(* PLC project Generated.project, CODESYS CODESYS V3.5 SP19 Patch 1 *)
(* stored: creationDateTime 2026-09-06T13:00:42.484991, modificationDateTime 2026-09-06T13:00:42.484991 *)

TYPE ST_Chain_Winch_Safety : STRUCT
  Idx301_EmergencyChainClosed : BOOL;  (* 1 = Boucle Urgence OK (Armé) | 0 = Arrêt d'Urgence Appuyé *)
  Idx302_SafeStopActive : BOOL;  (* 0 = Sain (Autorisé) | 1 = Arrêt Rapide Métier Actif *)
  Idx303_PowerCutOffActive : BOOL;  (* 0 = Puissance OK | 1 = Coupure Puissance Sécurité *)
  Idx304_TopSensorPhysical_DI : BOOL;  (* 1 = Capteur Haut Libre (Sain) | 0 = Butée Haute Atteinte *)
  Idx305_TopSensorBypassActive : BOOL;  (* 0 = Capteur Actif | 1 = Capteur Haut Shunté IHM ⚠️ *)
  Idx306_AscentPermitEffective : BOOL;  (* 1 = Ascending Autorisée | 0 = ASCENDING BLOQUÉE *)
  Idx307_SlackCablePhysical_DI : BOOL;  (* 1 = Câble Tendu (Sain) | 0 = Mou de Câble Détecté *)
  Idx308_SlackCableBypassActive : BOOL;  (* 0 = Capteur Actif | 1 = Mou de Câble Shunté IHM ⚠️ *)
  Idx309_DescendPermitEffective : BOOL;  (* 1 = Descending Autorisée | 0 = DESCENDING BLOQUÉE *)
  Idx310_ErrorOperatorComm : BOOL;  (* Défauts safety déchiffrés (bits ErrorId) — visibles individuellement à l'IHM bit0 Perte communication opérateur (joystick CAN / heartbeat IHM) *)
  Idx311_ErrorEncoder : BOOL;  (* bit1 Perte codeur de ce treuil *)
  Idx312_ErrorPhaseRotation : BOOL;  (* bit4 Mauvaise rotation de phases *)
  Idx313_ErrorMecaA : BOOL;  (* bit7 Mouvement non commandé / roue libre *)
  Idx314_ErrorMecaB : BOOL;  (* bit8 Absence confirmation arrêt sans commande *)
  Idx315_ErrorMecaC : BOOL;  (* bit9 Glissement M1 pendant cycle benne *)
  Idx316_ErrorMecaD : BOOL;  (* bit11 Non-arrêt sur capteur haut *)
  Idx317_ErrorMecaE : BOOL;  (* bit12/13 Écart synchro critique M1/M2 *)
  Idx318_ErrorBrakeThermal : BOOL;  (* bit10 Surchauffe thermique frein commun *)
  Idx319_ErrorOppositeDir : BOOL;  (* bit14 Sens réel opposé au sens commandé *)
  Idx320_ErrorNoMovement : BOOL;  (* bit15 Absence de mouvement malgré commande *)
  Idx321_CfgTopLimitM : REAL;  (* ⛔ Bloc "Pourquoi la montée ne s'arrête pas à la limite haute ?" — diagnostic ordonné (lecture maintenance) : config + position → butée atteinte → bypass actifs. 📐 Limite haute effective active (m) = CfgCableLimitAscent_M *)
  Idx322_CablePosM : REAL;  (* 📐 Position câble courante (m) *)
  Idx323_TopLimitReached : BOOL;  (* 1 = position >= limite haute (hors homing) | 0 = en dessous *)
  Idx324_AscentBlockedByTopLimit : BOOL;  (* 1 = montée réellement coupée par la butée logicielle (AscentPermit=0) | 0 = limitée non bloquante (bypass ?) *)
  Idx325_BypassTopLimitSoftware : BOOL;  (* ⚠️ 1 = butée logicielle shunétee IHM (individuel) *)
  Idx326_BypassTopLimitSoftCommun : BOOL;  (* ⚠️ 1 = butée logicielle shunétee (commun) *)
  Idx327_BypassTopLimitSwitch : BOOL;  (* ⚠️ 1 = capteur fin de course haut shuné IHM (individuel) *)
  Idx328_BypassTopLimitSwitchCommun : BOOL;  (* ⚠️ 1 = capteur fin de course haut shuné (commun) *)
  Idx329_BypassGlobal : BOOL;  (* ⚠️ 1 = bypass global treuil (individuel) *)
  Idx330_BypassGlobalCommun : BOOL;  (* ⚠️ 1 = bypass global (commun) *)
END_STRUCT;
END_TYPE
